// Block: A0304_Navetta_PERS

DATA_BLOCK A0304_Navetta_PERS
VERSION : 0.1
   NON_RETAIN
   VAR
      Par : Struct
         Ax_Man : Positioning_DOL_Machine_Par;
         Ax_Testa_Pers : Positioning_DOL_Machine_Pers_Data;
         Ax_Coda_Pers : Positioning_DOL_Machine_Pers_Data;
         Enc : Struct
            Testa : PosFbk_RTN;
            Coda : PosFbk_RTN;
         END_STRUCT;
      END_STRUCT;
      Par_Mach : Struct
         PosPrePrelievo : LReal;
         PosPrelievo : LReal;
         PosDeposito : LReal;
         ToleranceWindow : LReal;
      END_STRUCT;
   END_VAR

BEGIN
   // No initialization required
END_DATA_BLOCK
